PROGRAM PackML_02
VAR
	fbRobotCell			: FB_Cell_02;							// Unit, Machine Cell
	fbInfeed 			: FB_Infeed_02_01;						// SubUnit, Infeed Conveyor
	fbScara				: FB_Scara_02_02;						// SubUnit, Scara Robot
	fbDischarge			: FB_Discharge_02_03;					// SubUnit, Discharge Conveyor
	stPMLSubUnitInfo	: ARRAY [1..4] OF ST_PMLSubUnitInfo;	// Information about the Subunits
END_VAR

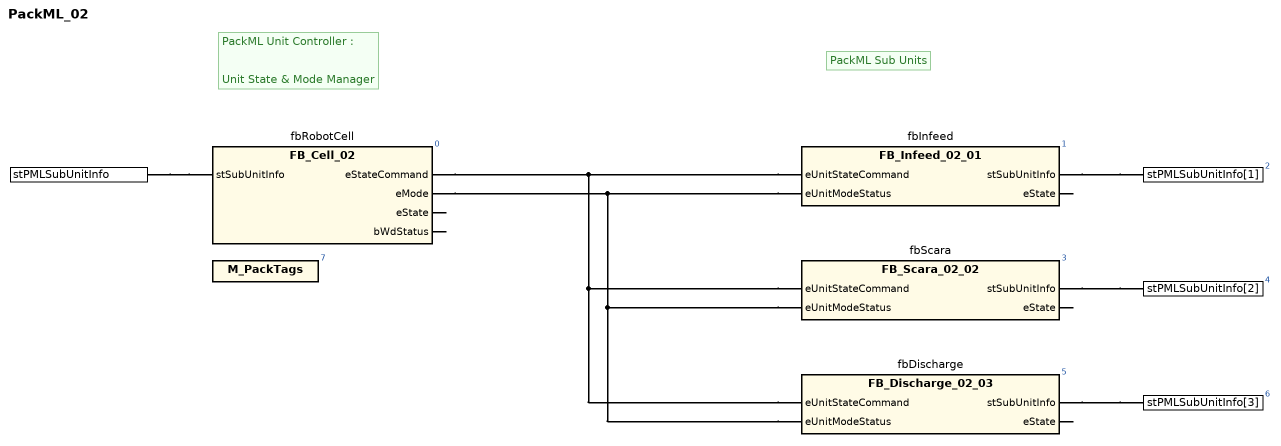
// PackML Unit Controller :
//
// Unit State & Mode Manager
fbRobotCell(stSubUnitInfo := stPMLSubUnitInfo); // FB_Cell_02
// PackML Sub Units
fbInfeed(eUnitStateCommand := fbRobotCell.eStateCommand, eUnitModeStatus := fbRobotCell.eMode); // FB_Infeed_02_01
stPMLSubUnitInfo[1] := fbInfeed.stSubUnitInfo;
fbScara(eUnitStateCommand := fbRobotCell.eStateCommand, eUnitModeStatus := fbRobotCell.eMode); // FB_Scara_02_02
stPMLSubUnitInfo[2] := fbScara.stSubUnitInfo;
fbDischarge(eUnitStateCommand := fbRobotCell.eStateCommand, eUnitModeStatus := fbRobotCell.eMode); // FB_Discharge_02_03
stPMLSubUnitInfo[3] := fbDischarge.stSubUnitInfo;
M_PackTags();

METHOD M_PackTags
VAR_INPUT
END_VAR


// Commands to Unit 02 from the Production Line
fbRobotCell.P_PackTags.Command := GVL.UnitPackTags[2].Command;

// Status & Admin Data of Unit 01 to the Production Line
GVL.UnitPackTags[2].Status	:= fbRobotCell.P_PackTags.Status;
GVL.UnitPackTags[2].Admin	:= fbRobotCell.P_PackTags.Admin;
END_METHOD

END_PROGRAM

(* stored: Version 1.1.0.1, ProductVersion 3.1.4024.11
   POU PackML_02: Id {5fab7823-76d2-44a1-a0a8-268ea7e9a805}, SpecialFunc None
   Method M_PackTags: Id {01275c3b-7e5f-4552-b91d-e2aed132be5f} *)
